// TIA Portal V17 export
// export: Created 2022-07-20T07:02:37.8396472Z, ExportSetting WithDefaults, DisplayName Totally Integrated Automation Portal, DisplayVersion V17, DisplayName TIA Portal Openness, DisplayVersion V17, DisplayName TIA Portal Version Control Interface, DisplayVersion V17, DisplayName SINAMICS Startdrive Advanced, DisplayVersion V17, DisplayName SINAMICS Startdrive G130, G150, S120, S150, SINAMICS MV, S210, DisplayVersion V17, DisplayName SINAMICS Startdrive G110M, G120, G120C, G120D, G120P, G115D, DisplayVersion V17, DisplayName STEP 7 Professional, DisplayVersion V17, DisplayName STEP 7 Safety, DisplayVersion V17, DisplayName WinCC Advanced, DisplayVersion V17
VAR_GLOBAL   // PLC tag table "CONSTANT_IFM_Devices"
END_VAR
VAR_GLOBAL CONSTANT   // user constants
   ID_BEACON_TOWER : Hw_Io := 501;
   PORT_BEACON_TOWER : Int := 2;
   ID_AL2301 : Hw_Io := 500;
   PORT_AL2301 : Int := 1;
   ID_AIR_MODULE_UNWINDER : Hw_Io := 358;
   PORT_AIR_MODULE_UNWINDER : Int := 3;
   ID_AIR_MODULE_REWINDER : Hw_Io := 474;
   PORT_AIR_MODULE_REWINDER : Int := 4;
   ID_SENSOR_DISTANCE_UNWINDER : Hw_Io := 360;
   PORT_SENSOR_DISTANCE_UNWINDER : Int := 5;
   ID_SENSOR_DISTANCE_REWINDER : Hw_Io := 464;
   PORT_SENSOR_DISTANCE_REWINDER : Int := 6;
END_VAR
